(* IEC 61131-3 sources: ctf1-cps6963/plc1, 4 files *)

(* ---- generated_plc1-defenses.st ---- *)
PROGRAM plc1
  VAR
    ColorSensor_RED AT %IW0 : INT;
    ColorSensor_GREEN AT %IW1 : INT;
    ColorSensor_BLUE AT %IW2 : INT;
    RangeSensor AT %IW3 : INT;
    Pump AT %QX0.4 : BOOL := False;
    treatmentComplete AT %IX100.0 : BOOL := False;
  END_VAR
  VAR
    desiredDistanceFill : REAL := 7.0;
    measuredDistance : REAL;
  END_VAR

  (*Workaround to distance measure bug*)
  measuredDistance := INT_TO_REAL(RangeSensor)/100.0;
  desiredDistanceFill := 7.0;

  (Defense: The plc will keep working until the finishing point)
  IF INT_TO_REAL(RangeSensor) > 0.0 and INT_TO_REAL(RangeSensor) < 99.0 THEN
    treatmentComplete := False;
  ELSE
    treatmentComplete := True;
  END_IF;

  IF treatmentComplete THEN
          IF measuredDistance > desiredDistanceFill THEN
            Pump := TRUE;
          ELSE
            Pump := FALSE;
          END_IF;
  END_IF;
END_PROGRAM

CONFIGURATION Config0

  RESOURCE Res0 ON PLC
    TASK task0(INTERVAL := T#20ms,PRIORITY := 0);
    PROGRAM instance0 WITH task0 : plc1;
  END_RESOURCE
END_CONFIGURATION

(* ---- generated_plc1.st ---- *)
PROGRAM plc1
  VAR
    ColorSensor_RED AT %IW0 : INT;
    ColorSensor_GREEN AT %IW1 : INT;
    ColorSensor_BLUE AT %IW2 : INT;
    RangeSensor AT %IW3 : INT;
    Pump AT %QX0.4 : BOOL := False;
    treatmentComplete AT %IX100.0 : BOOL := False;
  END_VAR
  VAR
    desiredDistanceFill : REAL := 7.0;
    measuredDistance : REAL;
  END_VAR

  (*Workaround to distance measure bug*)
  measuredDistance := INT_TO_REAL(RangeSensor)/100.0;
  desiredDistanceFill := 7.0;

  IF INT_TO_REAL(RangeSensor) > 99.0 THEN
    treatmentComplete := True;
  ELSE
    treatmentComplete := False;
  END_IF;

  IF treatmentComplete THEN
          IF measuredDistance > desiredDistanceFill THEN
            Pump := TRUE;
          ELSE
            Pump := FALSE;
          END_IF;
  END_IF;
END_PROGRAM

CONFIGURATION Config0

  RESOURCE Res0 ON PLC
    TASK task0(INTERVAL := T#20ms,PRIORITY := 0);
    PROGRAM instance0 WITH task0 : plc1;
  END_RESOURCE
END_CONFIGURATION

(* ---- malicious-attack1.st ---- *)
PROGRAM plc1
  VAR
    ColorSensor_RED AT %IW0 : INT;
    ColorSensor_GREEN AT %IW1 : INT;
    ColorSensor_BLUE AT %IW2 : INT;
    RangeSensor AT %IW3 : INT;
    Pump AT %QX0.4 : BOOL := False;
    treatmentComplete AT %IX100.0 : BOOL := False;
  END_VAR
  VAR
    desiredDistanceFill : REAL := 7.0;
    measuredDistance : REAL;
  END_VAR

  (*Workaround to distance measure bug*)
  measuredDistance := INT_TO_REAL(RangeSensor)/100.0;
  desiredDistanceFill := 7.0;

  (Attack: Stopping the plc before it starts)
  treatmentComplete := True;

  IF treatmentComplete THEN
          IF measuredDistance > desiredDistanceFill THEN
            Pump := TRUE;
          ELSE
            Pump := FALSE;
          END_IF;
  END_IF;
END_PROGRAM

CONFIGURATION Config0

  RESOURCE Res0 ON PLC
    TASK task0(INTERVAL := T#20ms,PRIORITY := 0);
    PROGRAM instance0 WITH task0 : plc1;
  END_RESOURCE
END_CONFIGURATION

(* ---- malicious-attack2.st ---- *)
PROGRAM plc1
  VAR
    ColorSensor_RED AT %IW1 : INT;
    ColorSensor_GREEN AT %IW2 : INT;
    ColorSensor_BLUE AT %IW3 : INT;
    RangeSensor AT %IW4 : INT;
    Pump AT %QX0.4 : BOOL := False;
    treatmentComplete AT %IX100.0 : BOOL := False;
  END_VAR
  VAR
    desiredDistanceFill : REAL := 7.0;
    measuredDistance : REAL;
  END_VAR

  (*Workaround to distance measure bug*)
  measuredDistance := INT_TO_REAL(1-RangeSensor)/100.0;
  desiredDistanceFill := 7.0;

  IF treatmentComplete THEN
          IF measuredDistance < desiredDistanceFill THEN
            Pump := TRUE;
          ELSE
            Pump := FALSE;
          END_IF;
  END_IF;
END_PROGRAM

CONFIGURATION Config0

  RESOURCE Res0 ON PLC
    TASK task0(INTERVAL := T#20ms,PRIORITY := 0);
    PROGRAM instance0 WITH task0 : plc1;
  END_RESOURCE
END_CONFIGURATION
